DATA_BLOCK "Station5UnLoadData"
{ S7_Optimized_Access := 'FALSE' }
VERSION : 0.1
NON_RETAIN
// ATTRIBUTES
// AUTO_NUMBER = False
// BLOCK_NUMBER = 519
// END_ATTRIBUTES
   STRUCT
      "PLC.PartTypeID" : Int;
      "PLC.Station5DMXCode" : String[50];
      "PLC.Station5RecipeNo" : Int;
      "PLC.PartStatus" : Int;
      "PLC.SubPartSN1" : String[50];
      "PLC.TransferTime" : String[50];
      "PLC.ShaftGlueIVPro" : Int;
      "PLC.ShaftGlueResult" : Int;
      "PLC.ShaftGlueIVScore1" : Int;
      "PLC.ShaftGlueIVScore2" : Int;
      "PLC.ShaftGlueIVScore3" : Int;
      "PLC.ShaftGlueIVScore4" : Int;
      "PLC.ShaftMagnetIVPro" : Int;
      "PLC.MagnetGlueResult" : Int;
      "PLC.MagnetIVScore" : Int;
      "PLC.GluePro" : Int;
      "PLC.NGCode" : Int;
      Spare_5 : Int;
      Spare_6 : Int;
      Spare_7 : Int;
      Spare_8 : Int;
      Spare_9 : Int;
      Spare_10 : Int;
      "MES.ErrorCode" : Int;
      "MES.ErrorMsg" : String[60];
   END_STRUCT;


BEGIN

END_DATA_BLOCK

